ACTION Up_31_Bahn_030201:
fbHardwareBahn030201(
	uiI_ProId								:= P_BahnHardware,
	uiI_TrEId_Sek_1							:= TrEId_030201_Roll1,
	uiI_TrEId_Sek_2							:= TrEId_030202_Roll2,
	uiI_AxId_Roll1							:= 0,
	uiI_AxId_Roll2							:= 0,
	uiI_AxId_Riem1							:= 0,
	uiI_FehlerId_Roll1						:= 4050,
	uiI_FehlerId_Roll2						:= 4150,
	uiI_FehlerId_Riem1						:= 4250,
	sI_Bahnname_Sek_1						:= '03.02.01',
	sI_Bahnname_Sek_2						:= '03.02.02',
	bI_Hand									:= fbEins[iEins_Id].OsHandEin,
	bI_Automatik							:= fbEins[iEins_Id].OsAutomatikEin,
	bI_Testbetrieb							:= gxTestbetriebOhneMaschineAktiv,
	bI_SicherheitOK							:= gxSicherheitsBereichQuittiertC[giSicher_C2_1],
	bI_FreigabeAutomatik					:= TRUE,
	bI_FreigabeHandVorZurueck_Roll1			:= astrGButtonManTransporte[ID_Bahn030201_Roll1].bSchalt,
	bI_FreigabeHandVorZurueck_Riem1			:= astrGButtonManTransporte[ID_Bahn030205_Riem].bSchalt,
	bI_FreigabeHandHebenSenkenSek1			:= astrGButtonManTransporte[ID_Bahn030201_Roll1].bSchalt
													OR astrGButtonManTransporte[ID_Bahn030205_Riem].bSchalt,
	bI_BahnDarfZurueckHand_Roll1			:= TRUE,
	bI_BahnDarfZurueckHand_Riem1			:= TRUE,
	bI_FreigabeHandVorZurueck_Roll2			:= astrGButtonManTransporte[ID_Bahn030202_Roll2].bSchalt,
	bI_FreigabeHandHebenSenkenSek2			:= astrGButtonManTransporte[ID_Bahn030202_Roll2].bSchalt
												OR astrGButtonManTransporte[ID_Bahn030205_Riem].bSchalt,
	bI_BahnDarfZurueckHand_Roll2			:= TRUE,
	bI_FreigabeReset						:= astrGButtonManTransporte[ID_Bahn030201_Roll1].bSchalt
												OR astrGButtonManTransporte[ID_Bahn030202_Roll2].bSchalt
												OR astrGButtonManTransporte[ID_Bahn030205_Riem].bSchalt,
	bI_StoerungAntrieb_Roll1				:= NOT fbG6UmrichterBahn030201_Roll1.bQ_Betriebsbereit
												and NOT fbG6UmrichterBahn030202_Roll2.bQ_Betriebsbereit,
	bI_Anfang_Roll1							:= NOT bIW302Transp11Anf
												OR NOT bIW302Transp12Anf,
	bI_Ende_Roll1							:= ( NOT bIW302Transp11TeilVorAnschl
												OR NOT bIW302Transp12TeilVorAnschl )
												AND ( strGHdshk_Bahn030201_Roll1.r_PosiRestwert_AufBahn = 0
													OR strGHdshk_Anschlag030201.b_Grundstellung ),
	bI_AufFoerderhoehe_Roll1				:= bIW302Transp2GS,
	bI_StoerungAntrieb_Roll2				:= NOT fbG6UmrichterBahn030203_Roll3.bQ_Betriebsbereit
												and NOT fbG6UmrichterBahn030204_Roll4.bQ_Betriebsbereit,
	bI_Anfang_Roll2							:= NOT bIW302Transp21Anf
												OR NOT bIW302Transp22Anf,
	bI_Ende_Roll2							:= ( NOT bIW302Transp21TeilVorAnschl
													OR NOT bIW302Transp22TeilVorAnschl )
												AND strGHdshk_Bahn030202_Roll2.r_PosiRestwert_AufBahn = 0,
	bI_AufFoerderhoehe_Roll2				:= bIW302Transp2GS,
	bI_StoerungAntrieb_Riem1				:= NOT fbG6UmrichterBahn030205_Riem.bQ_Betriebsbereit,
	bI_Anfang_Riem1							:= false,
	bI_Ende_Riem1							:= NOT bIW303Transp1AnfSpur1
												OR NOT bIW303Transp1AnfSpur2,
	bI_AufFoerderhoehe_Riem1				:= bIW302Transp2AS,
	bI_HebenSenkenInvers					:= FALSE,
	bI_VorZurueckInversHand					:= FALSE,
	bI_AbbruchPosi_AufBahn_Roll1			:= FALSE,
	bI_AbbruchPosi_AufBahn_Roll2			:= FALSE,
	bI_AbbruchPosi_AufBahn_Riem1			:= FALSE,
	bI_AbbruchPosi_VonBahn_Roll1			:= FALSE, 
	bI_AbbruchPosi_VonBahn_Roll2			:= FALSE ,
	bI_AbbruchPosi_VonBahn_Riem1			:= FALSE,
	bI_BahnenGrundSchnell_Sek_1				:= FALSE,
	bI_BahnenGrundSchnell_Sek_2				:= FALSE,
	bI_HubGrundWennFrei_Sek_1				:= FALSE,
	bI_HubGrundWennFrei_Sek_2				:= FALSE,
	bI_HubArbeitWennFrei_Sek_1				:= FALSE,
	bI_HubArbeitWennFrei_Sek_2				:= FALSE,
	bI_HubGrundWennBelegt_Sek_1				:= FALSE,
	bI_HubGrundWennBelegt_Sek_2				:= FALSE,
	bI_HubArbeitWennBelegt_Sek_1			:= FALSE,
	bI_HubArbeitWennBelegt_Sek_2			:= FALSE,
	bI_OhneSynchronVonBahn_Roll1			:= FALSE,
	bI_OhneSynchronVonBahn_Roll2			:= FALSE,
	bI_OhneSynchronVonBahn_Riem1			:= FALSE,
	bI_MitUeberwachungTeilNichtFreigegeben	:= FALSE,
	bI_NullkanteLangeTeileAufRolle2			:= TRUE,
	bI_ImpulsInit							:= bGImpulsInitSprache,
	bI_OhneImpulsgeber_Roll1				:= FALSE,
	bI_OhneImpulsgeber_Roll2				:= FALSE,
	bI_OhneImpulsgeber_Riem1				:= FALSE,
	strIO_GHdshk_Roll1						:= strGHdshk_Bahn030201_Roll1,
	strIO_GHdshk_Roll1_Vorg					:= strGHdshk_Bahn030101,
	strIO_GHdshk_Roll2						:= strGHdshk_Bahn030202_Roll2,
	strIO_GHdshk_Roll2_Nachf				:= strBahnaustausch_Leer,
	strIO_GHdshk_Riem1						:= strGHdshk_Bahn030205_Riem,
	strIO_GHdshk_Riem1_Vorg					:= strBahnaustausch_Leer,
	strIO_GHdshk_Riem1_Nachf				:= strGHdshk_Bahn030301,
	strIO_GLmHand							:= strGLmHand,
	strIO_TrE_Sek_1							:= GDat.TrE_Daten[TrEId_030201_Roll1],
	strIO_TrE_Sek_2							:= GDat.TrE_Daten[TrEId_030202_Roll2],
	strIO_Stoerungen						:= strGStoerungen[iEins_Id],
	bQ_Sektion1AS							=> ,
	bQ_Sektion2AS							=> ,
	bQ_Sektion1GS							=> ,
	bQ_Sektion2GS							=> );

(* Nur ein Hub für beide *)
	
	bQW302Transp2AS:= fbHardwareBahn030201.bQ_Sektion1AS;
	bQW302Transp2GS:= fbHardwareBahn030201.bQ_Sektion1GS;
	
fbG6UmrichterBahn030201_Roll1(
	sI_NetIDMaster						:= P_Ueberwachung_EtherCat.sNetId,
	sI_PfadXML							:= sGG6XMLPfad,
	sI_PfadSonderDatensatz				:= '',
	sI_Name								:= '=W302.EA11+S1-TA1',
	uiI_FxId							:= FxId_030201_Roll1,
	uiI_ProId							:= P_Umrichter,
	uiI_DevID							:= uiIDevID,
	diI_Statuswort						:= udiIW302TA11Statuswort,
	usiI_Umrichterstatus				:= usiIW302TA11UmrichterStatus,
	uiI_Datensatz						:= 1,
	iI_Istfrequenz						:= uiIW302TA11Istfrequenz,
	tI_ZeitBremse						:= t#500ms,
	rI_Beschleunigung					:= 0.1,
	rI_Verzoegerung						:= 0.1,
	rI_Sollgeschwindigkeit				:= ABS(strGHdshk_Bahn030201_Roll1.lr_Bahnspeed_Vorgabe),
	rI_Maxgeschwindigkeit				:= strGHdshk_Bahn030201_Roll1.str_BahnSpeed.rVmaxSpeed,
	bI_Aktiv							:= TRUE,
	bI_FehlerQuitt						:= strGLmHand.bI_QuittStoerung,
	bI_Testbetrieb						:= gxTestbetriebOhneMaschineAktiv,
	bI_StartUmrichter					:= gxSicherheitsBereichQuittiertC[giSicher_C2_1],
	bI_Reglerfreigabe					:= gxSicherheitsBereichVerzOKC[giSicher_C2_1],
	bI_DrehrichtungVor					:= strGHdshk_Bahn030201_Roll1.b_BahnVor,
	bI_DrehrichtungZurueck				:= strGHdshk_Bahn030201_Roll1.b_BahnZurueck,
	bI_EtherCATOK						:= P_Ueberwachung_EtherCat.xAlles_OK,
	bI_DrehInv							:= TRUE,
	uiQ_EtherCATAdresse					=> uiGEtherCATAdresse_KEB[FxId_030201_Roll1],
	iQ_Sollwert							=> uiQW302TA11Sollw,
	lrQ_Istwert							=> strGHdshk_Bahn030201_Roll1.lr_Bahnspeed_Ist,
	diQ_Control							=> udiQW302TA11Control,
	bQ_Betriebsbereit					=> ,
	bQ_BremseLoesen						=> bQW302Bremse11Loe,
	bQ_FehlerKEBDatenDownload			=> ,
	bQ_FehlerKeinIMAUmrichter			=> ,
	bQ_FehlerXMLDatei					=> ,
	bQ_FehlerParaLesen					=> ,
	bQ_FehlerParaSchreiben				=> ,
	bQ_FehlerAdresseLesen				=> ,
	strQ_Umrichterstatus				=> );

Aufruf_DisplayKEB.arI_DisplayKEB[FxId_030201_Roll1]:=
	fbG6UmrichterBahn030201_Roll1.strQ_Umrichterstatus.sConverterState;

fbG6UmrichterBahn030202_Roll2(
	sI_NetIDMaster						:= P_Ueberwachung_EtherCat.sNetId,
	sI_PfadXML							:= sGG6XMLPfad,
	sI_PfadSonderDatensatz				:= '',
	sI_Name								:= '=W302.EA12+S1-TA1',
	uiI_FxId							:= FxId_030202_Roll2,
	uiI_ProId							:= P_Umrichter,
	uiI_DevID							:= uiIDevID,
	diI_Statuswort						:= udiIW302TA12Statuswort,
	usiI_Umrichterstatus				:= usiIW302TA12UmrichterStatus,
	uiI_Datensatz						:= 1,
	iI_Istfrequenz						:= uiIW302TA12Istfrequenz,
	tI_ZeitBremse						:= t#500ms,
	rI_Beschleunigung					:= 0.1,
	rI_Verzoegerung						:= 0.1,
	rI_Sollgeschwindigkeit				:= ABS(strGHdshk_Bahn030201_Roll1.lr_Bahnspeed_Vorgabe),
	rI_Maxgeschwindigkeit				:= strGHdshk_Bahn030201_Roll1.str_BahnSpeed.rVmaxSpeed,
	bI_Aktiv							:= TRUE,
	bI_FehlerQuitt						:= strGLmHand.bI_QuittStoerung,
	bI_Testbetrieb						:= gxTestbetriebOhneMaschineAktiv,
	bI_StartUmrichter					:= gxSicherheitsBereichQuittiertC[giSicher_C2_1],
	bI_Reglerfreigabe					:= gxSicherheitsBereichVerzOKC[giSicher_C2_1],
	bI_DrehrichtungVor					:= strGHdshk_Bahn030201_Roll1.b_BahnVor,
	bI_DrehrichtungZurueck				:= strGHdshk_Bahn030201_Roll1.b_BahnZurueck,
	bI_EtherCATOK						:= P_Ueberwachung_EtherCat.xAlles_OK,
	bI_DrehInv							:= TRUE,
	uiQ_EtherCATAdresse					=> uiGEtherCATAdresse_KEB[FxId_030202_Roll2],
	iQ_Sollwert							=> uiQW302TA12Sollw,//uiQW302TA11Sollw,
	lrQ_Istwert							=> strGHdshk_Bahn030201_Roll1.lr_Bahnspeed_Ist,
	diQ_Control							=> udiQW302TA12Control,
	bQ_Betriebsbereit					=> ,
	bQ_BremseLoesen						=> bQW302Bremse12Loe,
	bQ_FehlerKEBDatenDownload			=> ,
	bQ_FehlerKeinIMAUmrichter			=> ,
	bQ_FehlerXMLDatei					=> ,
	bQ_FehlerParaLesen					=> ,
	bQ_FehlerParaSchreiben				=> ,
	bQ_FehlerAdresseLesen				=> ,
	strQ_Umrichterstatus				=> );

Aufruf_DisplayKEB.arI_DisplayKEB[FxId_030202_Roll2]:=
	fbG6UmrichterBahn030202_Roll2.strQ_Umrichterstatus.sConverterState;

fbG6UmrichterBahn030203_Roll3(
	sI_NetIDMaster						:= P_Ueberwachung_EtherCat.sNetId,
	sI_PfadXML							:= sGG6XMLPfad,
	sI_PfadSonderDatensatz				:= '',
	sI_Name								:= '=W302.EA21+S1-TA1',
	uiI_FxId							:= FxId_030203_Roll3,
	uiI_ProId							:= P_Umrichter,
	uiI_DevID							:= uiIDevID,
	diI_Statuswort						:= udiIW302TA21Statuswort,
	usiI_Umrichterstatus				:= usiIW302TA21UmrichterStatus,
	uiI_Datensatz						:= 1,
	iI_Istfrequenz						:= uiIW302TA21Istfrequenz,
	tI_ZeitBremse						:= t#500ms,
	rI_Beschleunigung					:= 0.1,
	rI_Verzoegerung						:= 0.1,
	rI_Sollgeschwindigkeit				:= ABS(strGHdshk_Bahn030202_Roll2.lr_Bahnspeed_Vorgabe),
	rI_Maxgeschwindigkeit				:= strGHdshk_Bahn030202_Roll2.str_BahnSpeed.rVmaxSpeed,
	bI_Aktiv							:= TRUE,
	bI_FehlerQuitt						:= strGLmHand.bI_QuittStoerung,
	bI_Testbetrieb						:= gxTestbetriebOhneMaschineAktiv,
	bI_StartUmrichter					:= gxSicherheitsBereichQuittiertC[giSicher_C2_1],
	bI_Reglerfreigabe					:= gxSicherheitsBereichVerzOKC[giSicher_C2_1],
	bI_DrehrichtungVor					:= strGHdshk_Bahn030202_Roll2.b_BahnVor,
	bI_DrehrichtungZurueck				:= strGHdshk_Bahn030202_Roll2.b_BahnZurueck,
	bI_EtherCATOK						:= P_Ueberwachung_EtherCat.xAlles_OK,
	bI_DrehInv							:= TRUE,
	uiQ_EtherCATAdresse					=> uiGEtherCATAdresse_KEB[FxId_030203_Roll3],
	iQ_Sollwert							=> uiQW302TA21Sollw,
	lrQ_Istwert							=> strGHdshk_Bahn030203_Roll3.lr_Bahnspeed_Ist,
	diQ_Control							=> udiQW302TA21Control,
	bQ_Betriebsbereit					=> ,
	bQ_BremseLoesen						=> bQW302Bremse21Loe,
	bQ_FehlerKEBDatenDownload			=> ,
	bQ_FehlerKeinIMAUmrichter			=> ,
	bQ_FehlerXMLDatei					=> ,
	bQ_FehlerParaLesen					=> ,
	bQ_FehlerParaSchreiben				=> ,
	bQ_FehlerAdresseLesen				=> ,
	strQ_Umrichterstatus				=> );

Aufruf_DisplayKEB.arI_DisplayKEB[FxId_030203_Roll3]:=
	fbG6UmrichterBahn030203_Roll3.strQ_Umrichterstatus.sConverterState;

fbG6UmrichterBahn030204_Roll4(
	sI_NetIDMaster						:= P_Ueberwachung_EtherCat.sNetId,
	sI_PfadXML							:= sGG6XMLPfad,
	sI_PfadSonderDatensatz				:= '',
	sI_Name								:= '=W302.EA22+S1-TA1',
	uiI_FxId							:= FxId_030204_Roll4,
	uiI_ProId							:= P_Umrichter,
	uiI_DevID							:= uiIDevID,
	diI_Statuswort						:= udiIW302TA22Statuswort,
	usiI_Umrichterstatus				:= usiIW302TA22UmrichterStatus,
	uiI_Datensatz						:= 1,
	iI_Istfrequenz						:= uiIW302TA22Istfrequenz,
	tI_ZeitBremse						:= t#500ms,
	rI_Beschleunigung					:= 0.1,
	rI_Verzoegerung						:= 0.1,
	rI_Sollgeschwindigkeit				:= ABS(strGHdshk_Bahn030202_Roll2.lr_Bahnspeed_Vorgabe),
	rI_Maxgeschwindigkeit				:= strGHdshk_Bahn030202_Roll2.str_BahnSpeed.rVmaxSpeed,
	bI_Aktiv							:= TRUE,
	bI_FehlerQuitt						:= strGLmHand.bI_QuittStoerung,
	bI_Testbetrieb						:= gxTestbetriebOhneMaschineAktiv,
	bI_StartUmrichter					:= gxSicherheitsBereichQuittiertC[giSicher_C2_1],
	bI_Reglerfreigabe					:= gxSicherheitsBereichVerzOKC[giSicher_C2_1],
	bI_DrehrichtungVor					:= strGHdshk_Bahn030202_Roll2.b_BahnVor,
	bI_DrehrichtungZurueck				:= strGHdshk_Bahn030202_Roll2.b_BahnZurueck,
	bI_EtherCATOK						:= P_Ueberwachung_EtherCat.xAlles_OK,
	bI_DrehInv							:= TRUE,
	uiQ_EtherCATAdresse					=> uiGEtherCATAdresse_KEB[FxId_030204_Roll4],
	iQ_Sollwert							=> uiQW302TA22Sollw,
	lrQ_Istwert							=> strGHdshk_Bahn030204_Roll4.lr_Bahnspeed_Ist,
	diQ_Control							=> udiQW302TA22Control,
	bQ_Betriebsbereit					=> ,
	bQ_BremseLoesen						=> bQW302Bremse22Loe,
	bQ_FehlerKEBDatenDownload			=> ,
	bQ_FehlerKeinIMAUmrichter			=> ,
	bQ_FehlerXMLDatei					=> ,
	bQ_FehlerParaLesen					=> ,
	bQ_FehlerParaSchreiben				=> ,
	bQ_FehlerAdresseLesen				=> ,
	strQ_Umrichterstatus				=> );

Aufruf_DisplayKEB.arI_DisplayKEB[FxId_030204_Roll4]:=
	fbG6UmrichterBahn030204_Roll4.strQ_Umrichterstatus.sConverterState;


	
fbG6UmrichterBahn030205_Riem(
	sI_NetIDMaster						:= P_Ueberwachung_EtherCat.sNetId,
	sI_PfadXML							:= sGG6XMLPfad,
	sI_PfadSonderDatensatz				:= '',
	sI_Name								:= '=W302.EB1+S1-TA1',
	uiI_FxId							:= FxId_030205_Riem,
	uiI_ProId							:= P_Umrichter,
	uiI_DevID							:= uiIDevID,
	diI_Statuswort						:= udiIW302TA1Statuswort,
	usiI_Umrichterstatus				:= usiIW302TA1UmrichterStatus,
	uiI_Datensatz						:= 1,
	iI_Istfrequenz						:= uiIW302TA1Istfrequenz,
	tI_ZeitBremse						:= t#500ms,
	rI_Beschleunigung					:= 0.1,
	rI_Verzoegerung						:= 0.1,
	rI_Sollgeschwindigkeit				:= ABS(strGHdshk_Bahn030205_Riem.lr_Bahnspeed_Vorgabe),
	rI_Maxgeschwindigkeit				:= strGHdshk_Bahn030205_Riem.str_BahnSpeed.rVmaxSpeed,
	bI_Aktiv							:= TRUE,
	bI_FehlerQuitt						:= strGLmHand.bI_QuittStoerung,
	bI_Testbetrieb						:= gxTestbetriebOhneMaschineAktiv,
	bI_StartUmrichter					:= gxSicherheitsBereichQuittiertC[giSicher_C2_1],
	bI_Reglerfreigabe					:= gxSicherheitsBereichVerzOKC[giSicher_C2_1],
	bI_DrehrichtungVor					:= strGHdshk_Bahn030205_Riem.b_BahnVor,
	bI_DrehrichtungZurueck				:= strGHdshk_Bahn030205_Riem.b_BahnZurueck,
	bI_EtherCATOK						:= P_Ueberwachung_EtherCat.xAlles_OK,
	bI_DrehInv							:= TRUE,
	uiQ_EtherCATAdresse					=> uiGEtherCATAdresse_KEB[FxId_030205_Riem],
	iQ_Sollwert							=> uiQW302TA1Sollw,
	lrQ_Istwert							=> strGHdshk_Bahn030205_Riem.lr_Bahnspeed_Ist,
	diQ_Control							=> udiQW302TA1Control,
	bQ_Betriebsbereit					=> ,
	bQ_BremseLoesen						=> ,
	bQ_FehlerKEBDatenDownload			=> ,
	bQ_FehlerKeinIMAUmrichter			=> ,
	bQ_FehlerXMLDatei					=> ,
	bQ_FehlerParaLesen					=> ,
	bQ_FehlerParaSchreiben				=> ,
	bQ_FehlerAdresseLesen				=> ,
	strQ_Umrichterstatus				=> );

Aufruf_DisplayKEB.arI_DisplayKEB[FxId_030205_Riem]:=
	fbG6UmrichterBahn030205_Riem.strQ_Umrichterstatus.sConverterState;

fbJobBahn030201(
	bI_MitPCJob_Sek_1							:= TRUE,
	bI_MitPCJob_Sek_2							:= TRUE,
	bI_FreigabeJobErzeugenSPS_Roll1_Vorg		:= FALSE,
	bI_FreigabeJobErzeugenSPS_Roll1_Roll2		:= FALSE,
	bI_FreigabeJobErzeugenSPS_Roll2_Roll1		:= FALSE,
	bI_FreigabeJobErzeugenSPS_Roll2_Nachf		:= FALSE,
	bI_FreigabeJobErzeugenSPS_Riem1_Vorg		:= FALSE,
	bI_FreigabeJobErzeugenSPS_Riem1_Nachf		:= FALSE,
	bI_FreigabeResetJob							:=	astrGButtonManTransporte[ID_Bahn030201_Roll1].bSchalt
														OR astrGButtonManTransporte[ID_Bahn030202_Roll2].bSchalt
														OR astrGButtonManTransporte[ID_Bahn030203_Roll3].bSchalt
														OR astrGButtonManTransporte[ID_Bahn030204_Roll4].bSchalt
														OR astrGButtonManTransporte[ID_Bahn030205_Riem].bSchalt,
	bI_FreigabeResetBahn						:=	astrGButtonManTransporte[ID_Bahn030201_Roll1].bSchalt
														OR astrGButtonManTransporte[ID_Bahn030202_Roll2].bSchalt
														OR astrGButtonManTransporte[ID_Bahn030203_Roll3].bSchalt
														OR astrGButtonManTransporte[ID_Bahn030204_Roll4].bSchalt
														OR astrGButtonManTransporte[ID_Bahn030205_Riem].bSchalt,
	bI_FreigabeFuerJob_Sek_1					:= bFreigabeFuerJob_C2_1,
	bI_ZusatzFreigabe_Sek_1						:= strGHdshk_Anschlag030201.b_Grundstellung
													OR ( strGHdshk_Bahn030202_Roll2.b_BahnBelegt
														AND GDat.TrE_Daten[TrEId_030202_Roll2].iAnzahlPlatten <> 0 ),
	bI_FreigabeFuerBuchen_Sek_1					:= bFreigabeFuerBuchen_C2_1,
	bI_FreigabeFuerJob_Sek_2					:= bFreigabeFuerJob_C2_1,
	bI_ZusatzFreigabe_Sek_2						:= strGHdshk_Anschlag030201.b_Grundstellung,
	bI_FreigabeFuerBuchen_Sek_2					:= bFreigabeFuerBuchen_C2_1,
	bI_MitAufBahnBeiVonBahn_Sek_1				:= FALSE,
	bI_MitAufBahnBeiVonBahn_Sek_2				:= FALSE,
	bI_Querfoerderer_Roll						:= FALSE,
	bI_Querfoerderer_Riem						:= FALSE,
	bI_BahnHKStop_Roll1							:= FALSE,
	bI_BahnHKStop_Roll2							:= FALSE,
	bI_BahnHKStop_Riem1							:= FALSE,
	bI_FreigabeAnBahnanfang_Roll1				:= FALSE,
	bI_FreigabeAnsBahnende_Roll1				:= strGHdshk_Anschlag030201.b_Arbeitsstellung, 
	bI_FreigabeAnBahnanfang_Roll2				:= FALSE,
	bI_FreigabeAnsBahnende_Roll2				:= FALSE, 
	bI_FreigabeAnBahnanfang_Riem1				:= FALSE,
	bI_FreigabeAnsBahnende_Riem1				:= FALSE,
	bI_Testbetrieb								:= gxTestbetriebOhneMaschineAktiv,
	bI_BeiResetJoblisteLoeschen					:= NOT bG3TecIstLeitsystem,
	bI_NullkanteLangeTeileAufRolle2				:= TRUE,
	uiI_ProId									:= P_BahnJob,
	iI_MaxAnzahlJobs_Sek_1						:= 1,
	iI_MaxAnzahlJobs_Sek_2						:= 1,
	diI_SperrenQuellBahnNrVonPortal				:= 0,
	diI_SperrenZielBahnNrVonPortal				:= 0,
	tI_Systemzeit								:= P_SystemzeitAuswerten.tDatumZeit_PC,
	strIO_GHdshk_Roll1							:= strGHdshk_Bahn030201_Roll1,
	strIO_GHdshk_Roll1_Vorg						:= strGHdshk_Bahn030101,
	strIO_GHdshk_Roll2							:= strGHdshk_Bahn030202_Roll2,
	strIO_GHdshk_Roll2_Nachf					:= strBahnaustausch_Leer,
	strIO_GHdshk_Riem1							:= strGHdshk_Bahn030205_Riem,
	strIO_GHdshk_Riem1_Vorg						:= strBahnaustausch_Leer,
	strIO_GHdshk_Riem1_Nachf					:= strGHdshk_Bahn030301,
	strIO_TrE_Sek_1								:= GDat.TrE_Daten[TrEId_030201_Roll1],
	strIO_TrE_Sek_2								:= GDat.TrE_Daten[TrEId_030202_Roll2],
	strIO_TrE_Roll_Vorg							:= GDat.TrE_Daten[TrEId_030101],
	strIO_TrE_Roll_Nachf						:= TrE_Daten_Leer,
	strIO_TrE_Riem1_Vorg						:= TrE_Daten_Leer,
	strIO_TrE_Riem1_Nachf						:= GDat.TrE_Daten[TrEId_030301],
	strIO_ArbTab_Job_Sek_1						:= GJobDat.ArbTab_Job[TrEId_030201_Roll1],
	strIO_ArbTab_Job_Sek_2						:= GJobDat.ArbTab_Job[TrEId_030202_Roll2],
	strIO_GLmHand								:= strGLmHand,
	bQ_GrundOK_Sek_1							=> ,
	bQ_GrundOK_Sek_2							=> ,
	bQ_ResetAktiv_Sek_1							=> ,
	bQ_ResetAktiv_Sek_2							=> );
END_ACTION

ACTION Up_32_Bahn_030101:

fbHardwareBahn030101(
	uiI_ProId							:= P_BahnHardware,
	uiI_TrEId							:= TrEId_030101,
	uiI_AxId							:= 0,
	uiI_FehlerId						:= 4000,
	sI_Bahnname							:= '03.01.01',
	bI_Hand								:= fbEins[iEins_Id].OsHandEin,
	bI_Automatik						:= fbEins[iEins_Id].OsAutomatikEin,
	bI_Testbetrieb						:= gxTestbetriebOhneMaschineAktiv,
	bI_SicherheitOK						:= gxSicherheitsBereichQuittiertC[giSicher_C1_1],
	bI_FreigabeAutomatik				:= TRUE,
	bI_FreigabeHandVorZurueck			:= astrGButtonManTransporte[ID_Bahn030101].bSchalt,
	bI_BahnDarfZurueckHand				:= FALSE,
	bI_FreigabeReset					:= astrGButtonManTransporte[ID_Bahn030101].bSchalt,
	bI_StoerungAntrieb					:= NOT fbG6UmrichterBahn030101.bQ_Betriebsbereit,
	bI_Anfang							:= FALSE,
	bI_BelegtKontrolle					:= FALSE,
	bI_Ende								:= NOT bIW302Transp11Anf
											OR NOT bIW302Transp12Anf,
	bI_VorZurueckInversHand				:= FALSE,
	bI_AbbruchPosi_AufBahn				:= FALSE,
	bI_AbbruchPosi_VonBahn				:= FALSE,
	bI_BahnenGrundSchnell				:= FALSE,
	bI_GrundZurueck						:= FALSE,
	bI_OhneSynchronVonBahn				:= FALSE,
	bI_NachlaufAmAnfangEnde				:= FALSE,
	bI_MitUeberwachungTeilNichtFreigegeben		:= FALSE,
	bI_ImpulsInit						:= bGImpulsInitSprache,
	bI_OhneImpulsgeber					:= FALSE,
	bI_AutoHandaufgabeAktiv				:= FALSE,
	bI_AutoHandentnahmeAktiv			:= FALSE,
	strIO_GHdshk						:= strGHdshk_Bahn030101,
	strIO_GHdshk_Vorg					:= strGHdshk_BahnExternW1,
	strIO_GHdshk_Nachf					:= strGHdshk_Bahn030201_Roll1,
	strIO_GLmHand						:= strGLmHand,
	strIO_TrE							:= GDat.TrE_Daten[TrEId_030101],
	strIO_Stoerungen					:= strGStoerungen[iEins_Id]);

fbG6UmrichterBahn030101(
	sI_NetIDMaster						:= P_Ueberwachung_EtherCat.sNetId,
	sI_PfadXML							:= sGG6XMLPfad,
	sI_PfadSonderDatensatz				:= '',
	sI_Name								:= '=W301.EA1+S1-TA1',
	uiI_FxId							:= FxId_030101,
	uiI_ProId							:= P_Umrichter,
	uiI_DevID							:= uiIDevID,
	diI_Statuswort						:= udiIW301TA1Statuswort,
	usiI_Umrichterstatus				:= usiIW301TA1UmrichterStatus,
	uiI_Datensatz						:= 1,
	iI_Istfrequenz						:= uiIW301TA1Istfrequenz,
	tI_ZeitBremse						:= t#500ms,
	rI_Beschleunigung					:= 0.1,
	rI_Verzoegerung						:= 0.1,
	rI_Sollgeschwindigkeit				:= LREAL_TO_REAL(ABS(strGHdshk_Bahn030101.lr_Bahnspeed_Vorgabe)),
	rI_Maxgeschwindigkeit				:= strGHdshk_Bahn030101.str_BahnSpeed.rVmaxSpeed,
	bI_Aktiv							:= TRUE,
	bI_FehlerQuitt						:= strGLmHand.bI_QuittStoerung,
	bI_Testbetrieb						:= gxTestbetriebOhneMaschineAktiv,
	bI_StartUmrichter					:= gxSicherheitsBereichQuittiertC[giSicher_C1_1],
	bI_Reglerfreigabe					:= gxSicherheitsBereichVerzOKC[giSicher_C1_1],
	bI_DrehrichtungVor					:= strGHdshk_Bahn030101.b_BahnVor,
	bI_DrehrichtungZurueck				:= strGHdshk_Bahn030101.b_BahnZurueck,
	bI_EtherCATOK						:= P_Ueberwachung_EtherCat.xAlles_OK,
	bI_DrehInv							:= TRUE,
	uiQ_EtherCATAdresse					=> uiGEtherCATAdresse_KEB[FxId_030101],
	iQ_Sollwert							=> uiQW301TA1Sollw,
	lrQ_Istwert							=> strGHdshk_Bahn030101.lr_Bahnspeed_Ist,
	diQ_Control							=> udiQW301TA1Control,
	bQ_Betriebsbereit					=> ,
	bQ_BremseLoesen						=> ,
	bQ_FehlerKEBDatenDownload			=> ,
	bQ_FehlerKeinIMAUmrichter			=> ,
	bQ_FehlerXMLDatei					=> ,
	bQ_FehlerParaLesen					=> ,
	bQ_FehlerParaSchreiben				=> ,
	bQ_FehlerAdresseLesen				=> ,
	strQ_Umrichterstatus				=> );

Aufruf_DisplayKEB.arI_DisplayKEB[FxId_030101]:=
	fbG6UmrichterBahn030101.strQ_Umrichterstatus.sConverterState;

fbJobBahn030101(
	bI_MitPCJob								:= TRUE,
	bI_FreigabeJobErzeugenSPS_Vorg			:= FALSE,
	bI_FreigabeJobErzeugenSPS_Nachf			:= FALSE,
	bI_FreigabeResetJob						:= astrGButtonManTransporte[ID_Bahn030101].bSchalt,
	bI_FreigabeResetBahn					:= astrGButtonManTransporte[ID_Bahn030101].bSchalt,
	bI_FreigabeFuerJob						:= bFreigabeFuerJob_C1_1,
	bI_ZusatzFreigabe						:= FALSE,
	bI_FreigabeFuerBuchen					:= bFreigabeFuerBuchen_C1_1,
	bI_MitAufBahnBeiVonBahn					:= FALSE,
	bI_Querfoerderer						:= FALSE,
	bI_FreigabeAnBahnanfang					:= FALSE,
	bI_FreigabeAnsBahnende					:= FALSE,
	bI_BilderSammeln						:= FALSE,
	bI_ScannenAktiv							:= FALSE,
	bI_Testbetrieb							:= gxTestbetriebOhneMaschineAktiv,
	bI_FehlerQuittScanner					:= FALSE,
	bI_BeiResetJoblisteLoeschen				:= NOT bG3TecIstLeitsystem,
	iI_MaxAnzahlJobs						:= 1,
	iI_MaxAnzahlNoRead						:= 1,
	uiI_ProId								:= P_BahnJob,
	diI_SperrenQuellBahnNrVonPortal			:= 0,
	diI_SperrenZielBahnNrVonPortal			:= 0,
	tI_BisScannerDatenDa					:= t#0s,
	tI_Systemzeit							:= P_SystemzeitAuswerten.tDatumZeit_PC,
	strIO_GHdshk							:= strGHdshk_Bahn030101,
	strIO_GHdshk_Vorg						:= strGHdshk_BahnExternW1,
	strIO_GHdshk_Nachf						:= strGHdshk_Bahn030201_Roll1,
	strIO_TrE								:= GDat.TrE_Daten[TrEId_030101],
	strIO_TrE_Vorg							:= GDat.TrE_Daten[TrEId_ExternW1],
	strIO_TrE_Nachf							:= GDat.TrE_Daten[TrEId_030201_Roll1],
	strIO_ArbTab_Job						:= GJobDat.ArbTab_Job[TrEId_030101],
	strIO_GLmHand							:= strGLmHand,
	fbIO_Scanner							:= fbScanner_Leer,
	bQ_GrundOK								=> ,
	bQ_ResetAktiv							=> ,
	bQ_ScannerHatNichtGelesen				=> ,
	bQ_ScannerFalscherBarcode				=> ,
	bQ_ScannerMaxAnzahlNoRead				=> );

(* Freigabe Ablegen *)
	
strGSignalaustauschExternW1.bQ_Vorgeschaltet_FreigabeAblegen:=
	GDat.TrE_Daten[TrEId_030101].iJobStatus = iDatenAktiv
	AND fbJobBahn030101.strBahnjob_Aktiv.diQuellId = strGHdshk_BahnExternW1.di_PlatzId
	AND fbJobBahn030101.strBahnjob_Aktiv.diZielId = strGHdshk_Bahn030101.di_PlatzId
	AND	GDat.TrE_Daten[TrEId_030101].iSperren = 0
	AND	GDat.TrE_Daten[TrEId_ExternW1].iSperren = 0
	AND	strGHdshk_Bahn030101.i_BahnV2_AufBahn_BereitFuerJob = 0
	AND	strGHdshk_Bahn030101.i_BahnV2_VonBahn_BereitFuerJob = 0
	AND	strGHdshk_Bahn030101.str_DoJob_AufBahn = eRolljobKeinJob
	AND	strGHdshk_Bahn030101.str_DoJob_VonBahn = eRolljobKeinJob
	AND	strGHdshk_Bahn030101.str_JobAktiv_AufBahn = eRolljobKeinJob
	AND	strGHdshk_Bahn030101.str_JobAktiv_VonBahn = eRolljobKeinJob
	AND	strGHdshk_Bahn030101.str_BahnStatus = iAutomatikBereitJob
	AND strGHdshk_Bahn030101.b_BahnSteht
	AND NOT strGHdshk_Bahn030101.b_BahnBelegt
	AND NOT strGHdshk_Bahn030101.b_LiAnfang
	AND NOT strGHdshk_Bahn030101.b_LiEnde
	AND	GDat.TrE_Daten[TrEId_030101].iAnzahlPlatten = 0
	AND	bFreigabeFuerJob_C1_1;

(* Jobhandling und Quittierung *)
		
IF GDat.TrE_Daten[TrEId_030101].iJobStatus = iDatenAktiv 
	AND strGSignalaustauschExternW1.bI_Vorgeschaltet_QuittWerkstueckAbgelegt
	AND NOT strGSignalaustauschExternW1.bQ_Vorgeschaltet_QuittWerkstueckAbgelegt
THEN

	F_ProtoText4( P_BahnJob, 'Bahn 03.01.01:Schelling - Platte abgelegt, Job an IPC beendet.', '', '', '' );
	strGSignalaustauschExternW1.bQ_Vorgeschaltet_QuittWerkstueckAbgelegt:= TRUE;

	(* BahnjobDaten in Ziel-TrE eintragen                                            *)
	(* iMode_Copy=2 (alle Platten an freier Stelle), iMode_Daten=0, Barcodeprüfung aus, Quelle, Ziel   *)
	fbJobDaten_In_ZielTrE(
		iMode_Copy:= 2,
		iMode_Daten:= 0,
		iBarcodePruefen:= 0,
		Jobzeile:= fbJobBahn030101.strBahnjob_Aktiv,
		TrE_Daten:= GDat.TrE_Daten[TrEId_030101] );

	(* Plattendaten verschieben Quell-TrE, dabei wird [1] gelöscht, wenn letztes Teil = TrE löschen *)
	fbDatenVerschieben_In_TrEDaten(
		iMode:= 0,
		iZeile:= 0,
		iAnzahl_Soll:= fbJobBahn030101.strBahnjob_Aktiv.iAnzahlPlatten,
		TrE_Daten:=  GDat.TrE_Daten[TrEId_ExternW1] );
		
	F_ProtoText4( P_BahnJob, 'Bahn 03.01.01: Schelling - Platte(n) abgelegt', ' - Barcode: ', GDat.TrE_Daten[TrEId_030101].asBarcode[1], '' );

	GDat.TrE_Daten[TrEId_030101].iJobStatus:= iQuittieren;

ELSIF NOT strGSignalaustauschExternW1.bI_Vorgeschaltet_QuittWerkstueckAbgelegt
	AND	strGSignalaustauschExternW1.bQ_Vorgeschaltet_QuittWerkstueckAbgelegt
	AND strGSignalaustauschExternW1.bI_Vorgeschaltet_LastaufnahmeAusStoerbereichAblegen 	// Portal muss erst rausfahren
THEN

	F_ProtoText4( P_BahnJob, 'Bahn 03.01.01: Quittierung durch Schelling - Platte abgelegt', '', '', '' );
	strGHdshk_Bahn030101.b_BahnBelegt:= TRUE;
	strGSignalaustauschExternW1.bQ_Vorgeschaltet_QuittWerkstueckAbgelegt:= FALSE;

END_IF

(* TrE-Status *)

IF NOT strGSignalaustauschExternW1.bI_Vorgeschaltet_MaschineFrei
	OR 	gxTestbetriebOhneMaschineAktiv
THEN
	GDat.TrE_Daten[TrEId_ExternW1].iBelegtStatus:= F_SetClearBelegtStatus ( TrEId_ExternW1, iSektionBelegt, TRUE );

	IF	strGSignalaustauschExternW2.bI_Vorgeschaltet_JobForward
		OR 	gxTestbetriebOhneMaschineAktiv
	THEN
		GDat.TrE_Daten[TrEId_ExternW1].iBelegtStatus:= F_SetClearBelegtStatus ( TrEId_ExternW1, iBereitFuerLader, TRUE );
	END_IF
ELSE
	GDat.TrE_Daten[TrEId_ExternW1].iBelegtStatus:= F_SetClearBelegtStatus ( TrEId_ExternW1, iSektionBelegt, FALSE );
	GDat.TrE_Daten[TrEId_ExternW1].iBelegtStatus:= F_SetClearBelegtStatus ( TrEId_ExternW1, iBereitFuerLader, FALSE );
END_IF;

IF ( NOT strGSignalaustauschExternW1.bI_Vorgeschaltet_SchutzOk
	OR NOT strGSignalaustauschExternW1.bI_Vorgeschaltet_SchutzVerzOk
	OR 	strGSignalaustauschExternW1.bI_Vorgeschaltet_Stoerung )
	AND NOT gxTestbetriebOhneMaschineAktiv
THEN
	GDat.TrE_Daten[TrEId_ExternW1].iAktivStatus:= iStoerung;

ELSIF strGSignalaustauschExternW1.bI_Vorgeschaltet_TippenAktiv
THEN
	GDat.TrE_Daten[TrEId_ExternW1].iAktivStatus:= iHand;

ELSIF strGSignalaustauschExternW1.bI_Vorgeschaltet_SchutzOk
	AND	strGSignalaustauschExternW1.bI_Vorgeschaltet_SchutzVerzOk
	//AND	strGSignalaustauschExternW1.bI_Vorgeschaltet_StartVorschub
	OR	gxTestbetriebOhneMaschineAktiv
THEN
	IF NOT strGSignalaustauschExternW1.bI_Vorgeschaltet_MaschineFrei
		//AND	strGSignalaustauschExternW1.bQ_Vorgeschaltet_VorschubAktiv
	THEN
		GDat.TrE_Daten[TrEId_ExternW1].iAktivStatus:= iAutomatikAktivJob;
	ELSE
		GDat.TrE_Daten[TrEId_ExternW1].iAktivStatus:= iAutomatikBereitJob;
		strGHdshk_BahnExternW1.str_BahnStatus:= iAutomatikBereitJob;
	END_IF;
ELSE
	GDat.TrE_Daten[TrEId_ExternW1].iAktivStatus:= 0;
END_IF;
END_ACTION

ACTION Up_90_Ausgaben:
(*----------------------------------------------*)
(*----------------------------------------------*)
(*          Bahnen oder Job's aktiv ?		*)
(*----------------------------------------------*)
(*----------------------------------------------*)


bQ_BereichJobAktiv_C1_1:=
	strGHdshk_Bahn030101.str_BahnStatus = iAutomatikAktivJob;

bQ_BereichJobAktiv_C2_1:=
	strGHdshk_Bahn030201_Roll1.str_BahnStatus = iAutomatikAktivJob
	OR	strGHdshk_Bahn030202_Roll2.str_BahnStatus = iAutomatikAktivJob
	OR	strGHdshk_Bahn030205_Riem.str_BahnStatus = iAutomatikAktivJob
	OR	strGHdshk_Bahn030301.str_BahnStatus = iAutomatikAktivJob
	OR	strGHdshk_Bahn030401.str_BahnStatus = iAutomatikAktivJob
	OR	strGHdshk_Bahn030501.str_BahnStatus = iAutomatikAktivJob
	OR	strGHdshk_Bahn030601.str_BahnStatus = iAutomatikAktivJob
	OR	strGHdshk_Bahn030701_Roll.str_BahnStatus = iAutomatikAktivJob
	OR	strGHdshk_Bahn030702_Riem1.str_BahnStatus = iAutomatikAktivJob
	OR	strGHdshk_Bahn030703_Riem2.str_BahnStatus = iAutomatikAktivJob
	OR	strGHdshk_Bahn031401.str_BahnStatus = iAutomatikAktivJob
	OR	strGHdshk_Bahn031501.str_BahnStatus = iAutomatikAktivJob
	OR	strGHdshk_Bahn032401.str_BahnStatus = iAutomatikAktivJob
	OR	strGHdshk_Bahn032501.str_BahnStatus = iAutomatikAktivJob
	OR	strGHdshk_Anschlag030201.str_ZylinderStatus = iAutomatikAktivJob
	OR	fbPosi_Wippe_030301.OwJobStatus = iAutomatikAktivJob
		AND NOT GKoAnWippe_030301.xAchse_Inaktiv
	OR	fbPosi_Wippe_030601.OwJobStatus = iAutomatikAktivJob
		AND NOT GKoAnWippe_030601.xAchse_Inaktiv;

bQ_BereichJobAktiv_C2_2:=
	strGHdshk_Bahn030801.str_BahnStatus = iAutomatikAktivJob;


(*----------------------------------------------*)
(*----------------------------------------------*)
(*       Bahnen und Job's beendet für		*)
(*                 Zyklusende ?			*)
(*----------------------------------------------*)
(*----------------------------------------------*)

bQ_BereichZyklusBeendet_C1_1:=
 	strGHdshk_Bahn030101.str_BahnStatus = iAutomatikBereitJob;

bQ_BereichZyklusBeendet_C2_1:=
 	strGHdshk_Bahn030201_Roll1.str_BahnStatus = iAutomatikBereitJob
 	AND strGHdshk_Bahn030202_Roll2.str_BahnStatus = iAutomatikBereitJob
 	AND strGHdshk_Bahn030205_Riem.str_BahnStatus = iAutomatikBereitJob
 	AND strGHdshk_Bahn030301.str_BahnStatus = iAutomatikBereitJob
 	AND strGHdshk_Bahn030401.str_BahnStatus = iAutomatikBereitJob
 	AND strGHdshk_Bahn030501.str_BahnStatus = iAutomatikBereitJob
 	AND strGHdshk_Bahn030601.str_BahnStatus = iAutomatikBereitJob
 	AND strGHdshk_Bahn030701_Roll.str_BahnStatus = iAutomatikBereitJob
 	AND strGHdshk_Bahn030702_Riem1.str_BahnStatus = iAutomatikBereitJob
 	AND strGHdshk_Bahn030703_Riem2.str_BahnStatus = iAutomatikBereitJob
 	AND strGHdshk_Bahn031401.str_BahnStatus = iAutomatikBereitJob
 	AND strGHdshk_Bahn031501.str_BahnStatus = iAutomatikBereitJob
 	AND strGHdshk_Bahn032401.str_BahnStatus = iAutomatikBereitJob
 	AND strGHdshk_Bahn032501.str_BahnStatus = iAutomatikBereitJob
	AND	strGHdshk_Anschlag030201.str_ZylinderStatus = iAutomatikBereitJob
	AND ( fbPosi_Wippe_030301.OwJobStatus = iAutomatikBereitJob
		AND	fbPosi_Wippe_030301.OsGrundstellungAchse
		AND	fbPosi_Wippe_030301.OsZyklusBeendet
		OR	bFreigabeTuerOeffnen_Wippe_030301
		OR	GKoAnWippe_030301.xAchse_Inaktiv )
	AND ( fbPosi_Wippe_030601.OwJobStatus = iAutomatikBereitJob
		AND	fbPosi_Wippe_030601.OsGrundstellungAchse
		AND	fbPosi_Wippe_030601.OsZyklusBeendet
		OR	bFreigabeTuerOeffnen_Wippe_030601
		OR	GKoAnWippe_030601.xAchse_Inaktiv );

bQ_BereichZyklusBeendet_C2_2:=
 	strGHdshk_Bahn030801.str_BahnStatus = iAutomatikBereitJob;


(*----------------------------------------------*)
(*----------------------------------------------*)
(*       Bahnen stehen					*)
(*----------------------------------------------*)
(*----------------------------------------------*)
bQ_BereichGestoppt_C1_1:=
	strGHdshk_Bahn030101.b_BahnSteht;
		
		
bQ_BereichGestoppt_C2_1:=
	strGHdshk_Bahn030201_Roll1.b_BahnSteht
	AND strGHdshk_Bahn030201_Roll1.b_BahnSteht
	AND strGHdshk_Bahn030202_Roll2.b_BahnSteht
	AND strGHdshk_Bahn030205_Riem.b_BahnSteht
	AND strGHdshk_Bahn030301.b_BahnSteht
	AND	strGHdshk_Bahn030401.b_BahnSteht
	AND	strGHdshk_Bahn030501.b_BahnSteht
	AND	strGHdshk_Bahn030601.b_BahnSteht
	AND	strGHdshk_Bahn030701_Roll.b_BahnSteht
	AND	strGHdshk_Bahn030702_Riem1.b_BahnSteht
	AND	strGHdshk_Bahn030703_Riem2.b_BahnSteht
	AND	strGHdshk_Bahn031401.b_BahnSteht
	AND	strGHdshk_Bahn031501.b_BahnSteht
	AND	strGHdshk_Bahn032401.b_BahnSteht
	AND	strGHdshk_Bahn032501.b_BahnSteht
	AND	strGHdshk_Anschlag030201.str_ZylinderStatus = iAutomatikBereitJob
	AND ( fbAchse_Wippe_030301.OwOut.xAchseBereit
		OR	fbAchse_Wippe_030301.OwOut.xAchseEnabled
		OR	fbAchse_Wippe_030301.OwOut.xAchseDisabled
		OR	GKoAnWippe_030301.xAchse_Inaktiv )
	AND ( fbAchse_Wippe_030601.OwOut.xAchseBereit
		OR	fbAchse_Wippe_030601.OwOut.xAchseEnabled
		OR	fbAchse_Wippe_030601.OwOut.xAchseDisabled
		OR	GKoAnWippe_030601.xAchse_Inaktiv );

bQ_BereichGestoppt_C2_2:=
	strGHdshk_Bahn030801.b_BahnSteht;


(*----------------------------------------------*)
(*----------------------------------------------*)
(*         Erkennung Stillstand			*)
(*----------------------------------------------*)
(*----------------------------------------------*)

bEineBahnBelegt:=
	strGHdshk_Bahn030101.b_BahnBelegt
	OR strGHdshk_Bahn030201_Roll1.b_BahnBelegt
	OR strGHdshk_Bahn030201_Roll1.b_BahnBelegt
	OR strGHdshk_Bahn030202_Roll2.b_BahnBelegt
	OR strGHdshk_Bahn030205_Riem.b_BahnBelegt
	OR strGHdshk_Bahn030301.b_BahnBelegt
	OR strGHdshk_Bahn030401.b_BahnSteht
	OR strGHdshk_Bahn030501.b_BahnBelegt
	OR strGHdshk_Bahn030601.b_BahnBelegt
	OR strGHdshk_Bahn030701_Roll.b_BahnBelegt
	OR strGHdshk_Bahn030702_Riem1.b_BahnSteht
	OR strGHdshk_Bahn030703_Riem2.b_BahnBelegt
	OR strGHdshk_Bahn031401.b_BahnBelegt
	OR strGHdshk_Bahn031501.b_BahnBelegt
	OR strGHdshk_Bahn032401.b_BahnBelegt
	OR strGHdshk_Bahn032501.b_BahnBelegt;

TBisErkennungStillstand.IN:=
	bQ_BereichZyklusBeendet_C1_1
	AND	bQ_BereichZyklusBeendet_C2_1
	AND	bQ_BereichZyklusBeendet_C2_2
	AND	bQ_BereichGestoppt_C1_1
	AND	bQ_BereichGestoppt_C2_1
	AND	bQ_BereichGestoppt_C2_2
	AND	bEineBahnBelegt
	AND	fbEins[iEins_Id].OsAutomatikStart
	AND	bFreigabeFuerJob_C1_1
	AND	bFreigabeFuerJob_C2_1
	AND	bFreigabeFuerJob_C2_2
	AND NOT strGStoerungen[iEins_Id].bStoerungDruckluft
	AND NOT strGStoerungen[iEins_Id].bAbsoluterStop
	AND NOT strGStoerungen[iEins_Id].bFehlerMitQuittung
	AND NOT strGStoerungen[iEins_Id].bBedingterStop
	AND NOT strGStoerungen[iEins_Id].bStoerungAntriebe
	AND NOT strGStoerungen[iEins_Id].bStoerungAblauf;

TBisErkennungStillstand( PT:= GKoAll.tBisErkennung_Stillstand );
bQ_MStillstand_TrotzBelegung:= TBisErkennungStillstand.Q;
END_ACTION

END_PROGRAM

(* stored: Version 1.1.0.1, ProductVersion 3.1.4024.12
   POU Aufruf_Eins_1_Bahnen_0301_Bis_0308: Id {b8d257ef-f671-462d-9c6d-78ad3fe4ceba}, SpecialFunc None
   Action Up_01_Meldungen: Id {44a06d00-3c2e-429b-a950-8e5aa5bb773f}
   Action Up_02_Reset_Grund_Freigabe: Id {a382013e-23ed-4c47-8640-78bf913e99d0}
   Action Up_10_AbsAchse_Wippe_030301: Id {d9c7d313-24d6-41c1-ae0b-bc89100aaab9}
   Action Up_11_AbsAchse_Posi_Wippe_030301: Id {e314877c-2bf8-4b29-96cf-4a3fb462cfc4}
   Action Up_12_AbsAchse_Wippe_030601: Id {53c27a87-0bbe-4421-ac06-31f6069540f0}
   Action Up_13_AbsAchse_Posi_Wippe_030601: Id {306470f6-ccf6-4916-a05a-7c1121aca135}
   Action Up_14_EilSchl_Buerste_030801: Id {fdbb3157-422e-4ece-89cf-8fb05ac28ee3}
   Action Up_15_EilSchl_PosiBuerste_030801: Id {95cff286-8dba-4323-ae18-692c9624bb18}
   Action Up_16_Anschlag_030201: Id {5026497d-32ea-4e16-bedb-a5a7932fdcee}
   Action Up_19_Bahn_040101_Extern: Id {7f7243d1-1b70-4ef4-8364-9b495b96daff}
   Action Up_21_Bahn_030801: Id {69b5b77c-8dda-4b29-80d1-61124a157f40}
   Action Up_22_Bahn_030701: Id {ced456a4-f4a5-4c44-8bf3-8ae1aa671b9c}
   Action Up_23_Bahn_030601: Id {f15e06cd-7317-40ac-afc9-fd4e73e365ae}
   Action Up_24_Bahn_032501: Id {5df1705f-23e7-44f1-9565-6ab8653422b0}
   Action Up_25_Bahn_032401: Id {9f9587cf-30ae-4442-9fe0-f358c9f1b81b}
   Action Up_26_Bahn_031501: Id {8139a2b4-c27f-4edd-8323-796654634328}
   Action Up_27_Bahn_031401: Id {a4b9da01-724f-4f7e-b537-377fa21c8f8f}
   Action Up_28_Bahn_030501: Id {8831c2a4-d856-4415-9e9d-4f0726e8c5c6}
   Action Up_29_Bahn_030401: Id {2d936456-18a7-4f83-9b31-97562463a4c1}
   Action Up_30_Bahn_030301: Id {6da63603-a52f-47bf-a285-ac0a3a622add}
   Action Up_31_Bahn_030201: Id {ab488a4c-81a8-4bdc-a082-21411fb53ed4}
   Action Up_32_Bahn_030101: Id {51c77241-185f-4640-accc-813151ca84e9}
   Action Up_90_Ausgaben: Id {9d6e3780-1a68-4e99-af59-a37faac82060} *)
